// Relays stopper state and sends a message when stopper state changes.
FUNCTION_BLOCK FB_StopperWatcher
VAR_INPUT
END_VAR
VAR_OUTPUT
END_VAR
VAR_IN_OUT
	stCurrentBP : ST_BeamParams;
END_VAR
VAR
    i_StopperOutLS AT %I* : BOOL;
    i_StopperInLS AT %I* : BOOL;

    q_StopperOUT_Relay AT %Q* : BOOL;
    q_StopperIN_Relay AT %Q* : BOOL;

    Stopper : UINT;
    StopperName : STRING;
	{attribute 'instance-path'}
    {attribute 'noinit'}
    sPath    :    T_MaxString;

    // Logging
    fbLogMsg : FB_LogMessage := (
        eSubSystem := E_Subsystem.MPS);

    rtIn : R_TRIG;
    rtOut : R_TRIG;

	bInit: BOOL := TRUE;
END_VAR

IF bInit THEN
	fbLogMsg.sJson := F_PMPS_JSON(StopperName, sPath, 1000);
	bInit := FALSE;
END_IF


rtIn(CLK := i_StopperInLS);
rtOut(CLK := i_StopperOutLS);

IF rtIn.Q THEN
    fbLogMsg.sMsg := CONCAT(StopperName, ' moved IN');
    fbLogMsg();
ELSIF rtOut.Q THEN
    fbLogMsg.sMsg := CONCAT(StopperName, ' moved OUT');
    fbLogMsg();
END_IF

q_StopperOUT_Relay := i_StopperOutLS;
q_StopperIN_Relay := i_StopperInLS;

// Update current beam parameters
stCurrentBP.aVetoDevices[Stopper] := i_StopperInLS;

END_FUNCTION_BLOCK

(* stored: Version 1.1.0.1, ProductVersion 3.1.4022.18
   POU FB_StopperWatcher: Id {a8ba1c9e-0ec9-4e64-9a98-24aa43e040d0}, SpecialFunc None *)
